// TwinCAT 3 PLC project Testing
// ProgramVersion: 3.1.4020.4
// libraries:
//   Tc2_Standard, * (Beckhoff Automation GmbH)
//   Tc2_System, * (Beckhoff Automation GmbH)
//   Tc2_Utilities, * (Beckhoff Automation GmbH)
//   Tc3_Module, * (Beckhoff Automation GmbH)
// project tree:
//   GVLs/ IOlinks.TcGVL
//   / PlcTask.TcTTO
//   POUs/BrowikLib/TimeFunction/ ReadTime.TcPOU
//   POUs/ MAIN.TcPOU
//   POUs/UC_Control/FBs/ Measurement.TcPOU
//   POUs/UC_Control/ UC_Measurements.TcPOU
// real-time tasks:
//   TASK PlcTask: cycle T#10ms, priority 20, ADS port 350
// I/O:
//   DEVICE Device 1 (CX9000-KBus)
//     Box 1 (CX9000-BK)
//   DEVICE Device 2 (CX-BK)
//     Box 2 (CX-BK)

CONFIGURATION Testing
    RESOURCE PLC ON TwinCAT3
        TASK PlcTask(INTERVAL := T#10ms, PRIORITY := 20);
        PROGRAM MAIN WITH PlcTask : MAIN;
    END_RESOURCE
END_CONFIGURATION

// ---- GVLs/IOlinks.TcGVL
{attribute 'qualified_only'}
VAR_GLOBAL
	
(*Variables for the first DI-card*)
	di01 AT %IX0.0 : BOOL;
	di02 AT %IX0.1 : BOOL;
	di03 AT %IX0.2 : BOOL;
	di04 AT %IX0.3 : BOOL;
	di05 AT %IX0.4 : BOOL;
	di06 AT %IX0.5 : BOOL;
	di07 AT %IX0.6 : BOOL;
	di08 AT %IX0.7 : BOOL;
	
END_VAR

// ---- POUs/MAIN.TcPOU
PROGRAM MAIN
VAR
END_VAR

VAR_INPUT
	diOne : bool; 
END_VAR

UC_Measurements();

END_PROGRAM

// ---- POUs/UC_Control/UC_Measurements.TcPOU
PROGRAM UC_Measurements
VAR
	Puls: BOOL;
	Value: DINT:= 100; 
	Adjustment: DINT:= 10000; 
	FlowMeter: Measurement;
END_VAR

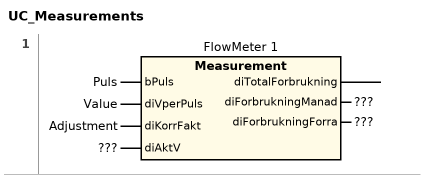
// NETWORK 1
FlowMeter 1(bPuls := Puls, diVperPuls := Value, diKorrFakt := Adjustment); // Measurement

END_PROGRAM

// ---- POUs/UC_Control/FBs/Measurement.TcPOU
FUNCTION_BLOCK Measurement
VAR_INPUT
	bPuls				: BOOL;
	diVperPuls			: DINT:= 10;	(*	Vad en puls är värd tex. 10 liter	*)
	diKorrFakt			: DINT:= 1000;	(*	Korrigeringsfaktor tex. pulserna är värde 10 liter men visningen ska vara m3 så ska denna faktor vara 1000	*)
END_VAR
VAR_OUTPUT
	diTotalForbrukning	: DINT;			(*	Den Totala Förbrukningen på Mätaren	*)
	diForbrukningManad	: DINT;			(*	Förbrukningen denna Månad	*)
	diForbrukningForra	: DINT;			(*	Förbrukningen Föregående Månad	*)
END_VAR
VAR_IN_OUT
	diAktV				: DINT;			(*	Aktuellt värde på mätaren	*)
END_VAR
VAR CONSTANT
	Jamnforelsedag		: STRING:='01'; 
END_VAR
VAR
	tidstring			: STRING;
	StringDag			: STRING;
	DagLika				: BOOL;
	Pf_Trig				: R_TRIG;
	PfTrigger			: R_TRIG;
	rAktV				: LREAL;
	rVperPuls			: LREAL;
	rKorrFakt			: LREAL;
	rTotalForbrukning	: LREAL;
	rTotalForbrukning1	: LREAL;
	rForbrukningForra	: LREAL;
	rForbrukningManad	: LREAL;
	ReadTime			: INT;
	Datum_Tid			: INT;
END_VAR

tidstring :=DT_TO_STRING(ReadTime.Datum_Tid);			(*Hej Hej*)
StringDag :=MID(tidstring,2,12); 						(*Välj position 12, och 2 höger/vänster inom char string, men frågan är vad som kommer ut från ReadTime.Datum_Tid*)

rAktV:=DINT_TO_LREAL( diAktV);
rVperPuls:=DINT_TO_LREAL (diVperPuls);
rKorrFakt:=DINT_TO_LREAL (diKorrFakt);

IF Jamnforelsedag = StringDag THEN  						(*Vad innebär det  dag "01" egentligen?!?*)
	DagLika:=TRUE;
ELSE
	DagLika:=FALSE;
END_IF

PfTrigger(CLK:=DagLika,); 									(*Kontrollerar om Daglika har blivit hög, och daglika är "01",  skulle tippa på att mätning samlas in en gång i månaden?*)
IF PfTrigger.Q THEN
	rForbrukningForra:=rForbrukningManad; 					(* Spara undan värdet för förra månaden*)
	rTotalForbrukning1:=rTotalForbrukning;	      			(* Sparar undan värdet för månaden eller veckan beroende på hur ofta dag 01 inträffar   *)
END_IF

Pf_Trig(CLK:= bPuls,);										(*Positiv Flankutvärdering på pulssignalen från givaren*)
IF Pf_Trig.Q THEN
	rAktV:=rAktV+rVperPuls;
	rTotalForbrukning:=rAktV/rKorrFakt;						(*Totalförbrukning för värdet just nu*)
END_IF

rForbrukningManad:=rTotalForbrukning-rTotalForbrukning1;	(*Beräknar förbrukning för den här månaden*)

(*Spara undan alla värden som  Dubbel INT*)

diAktV:=REAL_TO_DINT (rAktV);
diTotalForbrukning:=LREAL_TO_DINT (rTotalForbrukning);
diForbrukningForra:=LREAL_TO_DINT (rForbrukningForra);
diForbrukningManad:=LREAL_TO_DINT (rForbrukningManad);

END_FUNCTION_BLOCK

// ---- POUs/BrowikLib/TimeFunction/ReadTime.TcPOU
PROGRAM ReadTime
(*Utmaskning av Datum och Tid, används i Tidkanaler, Drifttidsmätnings-, Pulsmätnings funktionsblocken *)
VAR
	System_Tid	: NT_GetTime;
	Trigg		: TON;
	SysTime		: TIMESTRUCT;		(*	Denna variabel används av vissa funktionsblock som finns under Browik_FB	*)
	Datum_Tid	: DT; 				(*  Denna variabel används av vissa funktionsblock som finns under Browik_FB    *)
	Tid			: TOD; 				(*	Denna variabel i display WEBPORT för att visa lokal tid 					*)
	DayOfweek	: WORD; 			(*	Denna variabel används av vissa funktionsblock som finns under Browik_FB	*)
	Month		: WORD; 			(*	Denna variabel används av vissa funktionsblock som finns under Browik_FB	*)
	Day			: WORD;				(*	Denna variabel används av vissa funktionsblock som finns under Browik_FB	*)
END_VAR

Trigg(IN:= NOT Trigg.Q , PT:=T#1000MS , Q=> , ET=> );
System_Tid(START:=Trigg.Q );									(*Läsa in systemklockan vid positiv flank på signalen "Digital Input0"*)

Datum_Tid	:= SYSTEMTIME_TO_DT(System_Tid.TIMESTR);			(*Konvertera systemtid till datum och tid format*)
DayOfweek	:= System_Tid.TIMESTR.wDayOfWeek;					(*Läser ut veckodag ur sytemtiden*)
Month 		:= System_Tid.TIMESTR.wMonth;						(*Läder ut aktuell månad*)
Day  		:= System_Tid.TIMESTR.wDay;							(*Läser ut aktuell dag*)
SysTime		:= System_Tid.TIMESTR;								(*Läser ut hela TIMESTRUCTen*)
Tid 		:= DT_TO_TOD(Datum_Tid);							(*Läser ut aktuell tid*)

END_PROGRAM
